{attribute 'OPC.UA.DA' := '0'}
TYPE CalibratePMsConfig :
STRUCT
	LsCalibrateConfig : LsCalibrateConfig;
END_STRUCT
END_TYPE

(* stored: Version 1.1.0.1, ProductVersion 3.1.4024.3
   DUT CalibratePMsConfig: Id {4ceecc0f-f4aa-45c5-928e-90b392cf06df} *)
